(* IEC 61131-3 sources: RL_MAR/experiments/comparison/llm4plc/results/deepseek-ai-DeepSeek-V3.2_20260506_104945/20260506_120133, 4 files *)

(* ---- generated_code_iteration_0.st ---- *)
START_ST
FUNCTION_BLOCK CarParkingSystem
VAR_INPUT
    NewCarSlot : INT; (* Input for new car arrival slot number *)
END_VAR
VAR_OUTPUT
    Elevator1Busy : BOOL; (* Elevator 1 status - busy or idle *)
    Elevator2Busy : BOOL; (* Elevator 2 status - busy or idle *)
    Elevator1Position : INT; (* Elevator 1 current position *)
    Elevator2Position : INT; (* Elevator 2 current position *)
END_VAR
VAR
    Elevator1Target : INT; (* Elevator 1 target floor *)
    Elevator2Target : INT; (* Elevator 2 target floor *)
    CarSlots : ARRAY[1..100] OF BOOL; (* Array to represent parking slots - TRUE if occupied *)
    CurrentSlot : INT; (* Loop counter for scanning slots *)
    stateSys : INT; (* System state variable *)
    stateElev1 : INT; (* Elevator 1 state variable *)
    stateElev2 : INT; (* Elevator 2 state variable *)
    prevStateSys : INT; (* Previous system state for debugging or transitions *)
    prevStateElev1 : INT; (* Previous elevator 1 state *)
    prevStateElev2 : INT; (* Previous elevator 2 state *)
    tempSlot : INT; (* Temporary variable for processing new car slot *)
    movementStep : INT; (* Step size for elevator movement per cycle *)
    prevNewCarSlot : INT; (* Previous value of NewCarSlot for edge detection *)
    newArrivalDetected : BOOL; (* Flag to indicate a new arrival *)
    SYS_INIT : INT := 0; (* Constant for system initialization state *)
    SYS_SCAN : INT := 1; (* Constant for system scanning state *)
    ELEV_IDLE : INT := 0; (* Constant for elevator idle state *)
    ELEV_MOVING : INT := 1; (* Constant for elevator moving state *)
END_VAR

(* System state machine and elevator control logic *)
CASE stateSys OF
    SYS_INIT:
        (* Initialize all variables *)
        Elevator1Busy := FALSE;
        Elevator2Busy := FALSE;
        Elevator1Position := 0;
        Elevator2Position := 0;
        Elevator1Target := 0;
        Elevator2Target := 0;
        stateElev1 := ELEV_IDLE;
        stateElev2 := ELEV_IDLE;
        prevStateSys := SYS_INIT;
        prevStateElev1 := ELEV_IDLE;
        prevStateElev2 := ELEV_IDLE;
        tempSlot := 0;
        movementStep := 1;
        prevNewCarSlot := 0;
        newArrivalDetected := FALSE;
        FOR CurrentSlot := 1 TO 100 DO
            CarSlots[CurrentSlot] := FALSE;
        END_FOR;
        stateSys := SYS_SCAN; (* Transition to scanning state *)

    SYS_SCAN:
        (* Detect new car arrival by checking for change in NewCarSlot *)
        IF NewCarSlot <> prevNewCarSlot THEN
            newArrivalDetected := TRUE;
            prevNewCarSlot := NewCarSlot;
        ELSE
            newArrivalDetected := FALSE;
        END_IF;

        (* Process new arrival if detected and valid *)
        IF newArrivalDetected AND (NewCarSlot >= 1) AND (NewCarSlot <= 100) THEN
            IF NOT CarSlots[NewCarSlot] THEN
                CarSlots[NewCarSlot] := TRUE; (* Mark slot as occupied *)
                tempSlot := NewCarSlot;
                (* Assign target to appropriate elevator based on slot range *)
                IF (tempSlot >= 1) AND (tempSlot <= 50) THEN
                    (* Assign to Elevator 1 if idle *)
                    IF stateElev1 = ELEV_IDLE THEN
                        Elevator1Target := tempSlot;
                        stateElev1 := ELEV_MOVING;
                    END_IF;
                ELSIF (tempSlot >= 51) AND (tempSlot <= 100) THEN
                    (* Assign to Elevator 2 if idle *)
                    IF stateElev2 = ELEV_IDLE THEN
                        Elevator2Target := tempSlot;
                        stateElev2 := ELEV_MOVING;
                    END_IF;
                END_IF;
            END_IF;
        END_IF;

        (* Update Elevator 1 state and position *)
        CASE stateElev1 OF
            ELEV_IDLE:
                Elevator1Busy := FALSE;
                (* Position remains unchanged *)

            ELEV_MOVING:
                Elevator1Busy := TRUE;
                (* Move towards target by movementStep per cycle *)
                IF Elevator1Position < Elevator1Target THEN
                    Elevator1Position := Elevator1Position + movementStep;
                    IF Elevator1Position > Elevator1Target THEN
                        Elevator1Position := Elevator1Target;
                    END_IF;
                ELSIF Elevator1Position > Elevator1Target THEN
                    Elevator1Position := Elevator1Position - movementStep;
                    IF Elevator1Position < Elevator1Target THEN
                        Elevator1Position := Elevator1Target;
                    END_IF;
                END_IF;
                (* Check if target reached *)
                IF Elevator1Position = Elevator1Target THEN
                    stateElev1 := ELEV_IDLE;
                END_IF;
        END_CASE;

        (* Update Elevator 2 state and position *)
        CASE stateElev2 OF
            ELEV_IDLE:
                Elevator2Busy := FALSE;
                (* Position remains unchanged *)

            ELEV_MOVING:
                Elevator2Busy := TRUE;
                (* Move towards target by movementStep per cycle *)
                IF Elevator2Position < Elevator2Target THEN
                    Elevator2Position := Elevator2Position + movementStep;
                    IF Elevator2Position > Elevator2Target THEN
                        Elevator2Position := Elevator2Target;
                    END_IF;
                ELSIF Elevator2Position > Elevator2Target THEN
                    Elevator2Position := Elevator2Position - movementStep;
                    IF Elevator2Position < Elevator2Target THEN
                        Elevator2Position := Elevator2Target;
                    END_IF;
                END_IF;
                (* Check if target reached *)
                IF Elevator2Position = Elevator2Target THEN
                    stateElev2 := ELEV_IDLE;
                END_IF;
        END_CASE;

        (* Store previous states for potential debugging *)
        prevStateSys := stateSys;
        prevStateElev1 := stateElev1;
        prevStateElev2 := stateElev2;

        (* System remains in scanning state *)
        stateSys := SYS_SCAN;

END_CASE;

END_FUNCTION_BLOCK
END_ST

(* ---- generated_code_iteration_1.st ---- *)
START_REASON
The validation feedback indicates a CODESYS compiler error: "CASE标号要求文字或符号整型常量". This translates to "CASE label requires a literal or symbolic integer constant." This error occurs because in the provided ST code, the CASE statement for `stateSys` uses variables `SYS_INIT` and `SYS_SCAN` as case labels, but these are declared as variables within the VAR section with initial values (e.g., `SYS_INIT : INT := 0;`). In CODESYS, CASE labels must be constants (literals like 0, 1, or symbolic constants defined with `CONSTANT`), not variables. Variables cannot be used as case labels because their values can change at runtime, which is not allowed for case selection. To fix this, I need to declare `SYS_INIT`, `SYS_SCAN`, `ELEV_IDLE`, and `ELEV_MOVING` as constants using the `CONSTANT` keyword in a separate VAR_CONSTANT section, ensuring they are immutable and can be used as case labels. Additionally, I should ensure proper variable declarations and maintain the FUNCTION_BLOCK structure as required.
END_REASON

START_ST
FUNCTION_BLOCK CarParkingSystem
VAR_INPUT
    NewCarSlot : INT; (* Input for new car arrival slot number *)
END_VAR
VAR_OUTPUT
    Elevator1Busy : BOOL; (* Elevator 1 status - busy or idle *)
    Elevator2Busy : BOOL; (* Elevator 2 status - busy or idle *)
    Elevator1Position : INT; (* Elevator 1 current position *)
    Elevator2Position : INT; (* Elevator 2 current position *)
END_VAR
VAR
    Elevator1Target : INT; (* Elevator 1 target floor *)
    Elevator2Target : INT; (* Elevator 2 target floor *)
    CarSlots : ARRAY[1..100] OF BOOL; (* Array to represent parking slots - TRUE if occupied *)
    CurrentSlot : INT; (* Loop counter for scanning slots *)
    stateSys : INT; (* System state variable *)
    stateElev1 : INT; (* Elevator 1 state variable *)
    stateElev2 : INT; (* Elevator 2 state variable *)
    prevStateSys : INT; (* Previous system state for debugging or transitions *)
    prevStateElev1 : INT; (* Previous elevator 1 state *)
    prevStateElev2 : INT; (* Previous elevator 2 state *)
    tempSlot : INT; (* Temporary variable for processing new car slot *)
    movementStep : INT; (* Step size for elevator movement per cycle *)
    prevNewCarSlot : INT; (* Previous value of NewCarSlot for edge detection *)
    newArrivalDetected : BOOL; (* Flag to indicate a new arrival *)
END_VAR
VAR_CONSTANT
    SYS_INIT : INT := 0; (* Constant for system initialization state *)
    SYS_SCAN : INT := 1; (* Constant for system scanning state *)
    ELEV_IDLE : INT := 0; (* Constant for elevator idle state *)
    ELEV_MOVING : INT := 1; (* Constant for elevator moving state *)
END_VAR

(* System state machine and elevator control logic *)
CASE stateSys OF
    SYS_INIT:
        (* Initialize all variables *)
        Elevator1Busy := FALSE;
        Elevator2Busy := FALSE;
        Elevator1Position := 0;
        Elevator2Position := 0;
        Elevator1Target := 0;
        Elevator2Target := 0;
        stateElev1 := ELEV_IDLE;
        stateElev2 := ELEV_IDLE;
        prevStateSys := SYS_INIT;
        prevStateElev1 := ELEV_IDLE;
        prevStateElev2 := ELEV_IDLE;
        tempSlot := 0;
        movementStep := 1;
        prevNewCarSlot := 0;
        newArrivalDetected := FALSE;
        FOR CurrentSlot := 1 TO 100 DO
            CarSlots[CurrentSlot] := FALSE;
        END_FOR;
        stateSys := SYS_SCAN; (* Transition to scanning state *)

    SYS_SCAN:
        (* Detect new car arrival by checking for change in NewCarSlot *)
        IF NewCarSlot <> prevNewCarSlot THEN
            newArrivalDetected := TRUE;
            prevNewCarSlot := NewCarSlot;
        ELSE
            newArrivalDetected := FALSE;
        END_IF;

        (* Process new arrival if detected and valid *)
        IF newArrivalDetected AND (NewCarSlot >= 1) AND (NewCarSlot <= 100) THEN
            IF NOT CarSlots[NewCarSlot] THEN
                CarSlots[NewCarSlot] := TRUE; (* Mark slot as occupied *)
                tempSlot := NewCarSlot;
                (* Assign target to appropriate elevator based on slot range *)
                IF (tempSlot >= 1) AND (tempSlot <= 50) THEN
                    (* Assign to Elevator 1 if idle *)
                    IF stateElev1 = ELEV_IDLE THEN
                        Elevator1Target := tempSlot;
                        stateElev1 := ELEV_MOVING;
                    END_IF;
                ELSIF (tempSlot >= 51) AND (tempSlot <= 100) THEN
                    (* Assign to Elevator 2 if idle *)
                    IF stateElev2 = ELEV_IDLE THEN
                        Elevator2Target := tempSlot;
                        stateElev2 := ELEV_MOVING;
                    END_IF;
                END_IF;
            END_IF;
        END_IF;

        (* Update Elevator 1 state and position *)
        CASE stateElev1 OF
            ELEV_IDLE:
                Elevator1Busy := FALSE;
                (* Position remains unchanged *)

            ELEV_MOVING:
                Elevator1Busy := TRUE;
                (* Move towards target by movementStep per cycle *)
                IF Elevator1Position < Elevator1Target THEN
                    Elevator1Position := Elevator1Position + movementStep;
                    IF Elevator1Position > Elevator1Target THEN
                        Elevator1Position := Elevator1Target;
                    END_IF;
                ELSIF Elevator1Position > Elevator1Target THEN
                    Elevator1Position := Elevator1Position - movementStep;
                    IF Elevator1Position < Elevator1Target THEN
                        Elevator1Position := Elevator1Target;
                    END_IF;
                END_IF;
                (* Check if target reached *)
                IF Elevator1Position = Elevator1Target THEN
                    stateElev1 := ELEV_IDLE;
                END_IF;
        END_CASE;

        (* Update Elevator 2 state and position *)
        CASE stateElev2 OF
            ELEV_IDLE:
                Elevator2Busy := FALSE;
                (* Position remains unchanged *)

            ELEV_MOVING:
                Elevator2Busy := TRUE;
                (* Move towards target by movementStep per cycle *)
                IF Elevator2Position < Elevator2Target THEN
                    Elevator2Position := Elevator2Position + movementStep;
                    IF Elevator2Position > Elevator2Target THEN
                        Elevator2Position := Elevator2Target;
                    END_IF;
                ELSIF Elevator2Position > Elevator2Target THEN
                    Elevator2Position := Elevator2Position - movementStep;
                    IF Elevator2Position < Elevator2Target THEN
                        Elevator2Position := Elevator2Target;
                    END_IF;
                END_IF;
                (* Check if target reached *)
                IF Elevator2Position = Elevator2Target THEN
                    stateElev2 := ELEV_IDLE;
                END_IF;
        END_CASE;

        (* Store previous states for potential debugging *)
        prevStateSys := stateSys;
        prevStateElev1 := stateElev1;
        prevStateElev2 := stateElev2;

        (* System remains in scanning state *)
        stateSys := SYS_SCAN;

END_CASE;

END_FUNCTION_BLOCK
END_ST

(* ---- generated_code_iteration_2.st ---- *)
START_REASON
The validation feedback indicates an encoding issue: "gbk codec can't decode byte 0xac in position 101: illegal multibyte sequence." This suggests that the ST code contains a character that cannot be decoded with the GBK encoding, likely due to a special character like a non-breaking space, curly quotes, or an em dash that was inadvertently included. This could have been introduced in the previous response, possibly from copying or formatting. To fix this, I need to ensure the code uses only ASCII characters or properly encoded UTF-8 characters if supported, but for safety, I'll stick to basic ASCII characters (e.g., standard quotes, spaces, and alphanumeric symbols). I'll regenerate the code from scratch, ensuring no special or invisible characters are present, and maintain the FUNCTION_BLOCK structure with constants in VAR_CONSTANT as previously corrected. I'll also verify that all syntax is correct for CODESYS, including proper use of CASE statements with constants.
END_REASON

START_ST
FUNCTION_BLOCK CarParkingSystem
VAR_INPUT
    NewCarSlot : INT; (* Input for new car arrival slot number *)
END_VAR
VAR_OUTPUT
    Elevator1Busy : BOOL; (* Elevator 1 status - busy or idle *)
    Elevator2Busy : BOOL; (* Elevator 2 status - busy or idle *)
    Elevator1Position : INT; (* Elevator 1 current position *)
    Elevator2Position : INT; (* Elevator 2 current position *)
END_VAR
VAR
    Elevator1Target : INT; (* Elevator 1 target floor *)
    Elevator2Target : INT; (* Elevator 2 target floor *)
    CarSlots : ARRAY[1..100] OF BOOL; (* Array to represent parking slots - TRUE if occupied *)
    CurrentSlot : INT; (* Loop counter for scanning slots *)
    stateSys : INT; (* System state variable *)
    stateElev1 : INT; (* Elevator 1 state variable *)
    stateElev2 : INT; (* Elevator 2 state variable *)
    prevStateSys : INT; (* Previous system state for debugging or transitions *)
    prevStateElev1 : INT; (* Previous elevator 1 state *)
    prevStateElev2 : INT; (* Previous elevator 2 state *)
    tempSlot : INT; (* Temporary variable for processing new car slot *)
    movementStep : INT; (* Step size for elevator movement per cycle *)
    prevNewCarSlot : INT; (* Previous value of NewCarSlot for edge detection *)
    newArrivalDetected : BOOL; (* Flag to indicate a new arrival *)
END_VAR
VAR_CONSTANT
    SYS_INIT : INT := 0; (* Constant for system initialization state *)
    SYS_SCAN : INT := 1; (* Constant for system scanning state *)
    ELEV_IDLE : INT := 0; (* Constant for elevator idle state *)
    ELEV_MOVING : INT := 1; (* Constant for elevator moving state *)
END_VAR

(* System state machine and elevator control logic *)
CASE stateSys OF
    SYS_INIT:
        (* Initialize all variables *)
        Elevator1Busy := FALSE;
        Elevator2Busy := FALSE;
        Elevator1Position := 0;
        Elevator2Position := 0;
        Elevator1Target := 0;
        Elevator2Target := 0;
        stateElev1 := ELEV_IDLE;
        stateElev2 := ELEV_IDLE;
        prevStateSys := SYS_INIT;
        prevStateElev1 := ELEV_IDLE;
        prevStateElev2 := ELEV_IDLE;
        tempSlot := 0;
        movementStep := 1;
        prevNewCarSlot := 0;
        newArrivalDetected := FALSE;
        FOR CurrentSlot := 1 TO 100 DO
            CarSlots[CurrentSlot] := FALSE;
        END_FOR;
        stateSys := SYS_SCAN; (* Transition to scanning state *)

    SYS_SCAN:
        (* Detect new car arrival by checking for change in NewCarSlot *)
        IF NewCarSlot <> prevNewCarSlot THEN
            newArrivalDetected := TRUE;
            prevNewCarSlot := NewCarSlot;
        ELSE
            newArrivalDetected := FALSE;
        END_IF;

        (* Process new arrival if detected and valid *)
        IF newArrivalDetected AND (NewCarSlot >= 1) AND (NewCarSlot <= 100) THEN
            IF NOT CarSlots[NewCarSlot] THEN
                CarSlots[NewCarSlot] := TRUE; (* Mark slot as occupied *)
                tempSlot := NewCarSlot;
                (* Assign target to appropriate elevator based on slot range *)
                IF (tempSlot >= 1) AND (tempSlot <= 50) THEN
                    (* Assign to Elevator 1 if idle *)
                    IF stateElev1 = ELEV_IDLE THEN
                        Elevator1Target := tempSlot;
                        stateElev1 := ELEV_MOVING;
                    END_IF;
                ELSIF (tempSlot >= 51) AND (tempSlot <= 100) THEN
                    (* Assign to Elevator 2 if idle *)
                    IF stateElev2 = ELEV_IDLE THEN
                        Elevator2Target := tempSlot;
                        stateElev2 := ELEV_MOVING;
                    END_IF;
                END_IF;
            END_IF;
        END_IF;

        (* Update Elevator 1 state and position *)
        CASE stateElev1 OF
            ELEV_IDLE:
                Elevator1Busy := FALSE;
                (* Position remains unchanged *)

            ELEV_MOVING:
                Elevator1Busy := TRUE;
                (* Move towards target by movementStep per cycle *)
                IF Elevator1Position < Elevator1Target THEN
                    Elevator1Position := Elevator1Position + movementStep;
                    IF Elevator1Position > Elevator1Target THEN
                        Elevator1Position := Elevator1Target;
                    END_IF;
                ELSIF Elevator1Position > Elevator1Target THEN
                    Elevator1Position := Elevator1Position - movementStep;
                    IF Elevator1Position < Elevator1Target THEN
                        Elevator1Position := Elevator1Target;
                    END_IF;
                END_IF;
                (* Check if target reached *)
                IF Elevator1Position = Elevator1Target THEN
                    stateElev1 := ELEV_IDLE;
                END_IF;
        END_CASE;

        (* Update Elevator 2 state and position *)
        CASE stateElev2 OF
            ELEV_IDLE:
                Elevator2Busy := FALSE;
                (* Position remains unchanged *)

            ELEV_MOVING:
                Elevator2Busy := TRUE;
                (* Move towards target by movementStep per cycle *)
                IF Elevator2Position < Elevator2Target THEN
                    Elevator2Position := Elevator2Position + movementStep;
                    IF Elevator2Position > Elevator2Target THEN
                        Elevator2Position := Elevator2Target;
                    END_IF;
                ELSIF Elevator2Position > Elevator2Target THEN
                    Elevator2Position := Elevator2Position - movementStep;
                    IF Elevator2Position < Elevator2Target THEN
                        Elevator2Position := Elevator2Target;
                    END_IF;
                END_IF;
                (* Check if target reached *)
                IF Elevator2Position = Elevator2Target THEN
                    stateElev2 := ELEV_IDLE;
                END_IF;
        END_CASE;

        (* Store previous states for potential debugging *)
        prevStateSys := stateSys;
        prevStateElev1 := stateElev1;
        prevStateElev2 := stateElev2;

        (* System remains in scanning state *)
        stateSys := SYS_SCAN;

END_CASE;

END_FUNCTION_BLOCK
END_ST

(* ---- generated_code_iteration_3.st ---- *)
START_REASON
The validation feedback indicates a CODESYS compiler error: "应该采用VAR, VAR_INPUT, VAR_OUTPUT 或 VAR_IN_OUT 取代VAR_CONSTANT:;" which translates to "Should use VAR, VAR_INPUT, VAR_OUTPUT or VAR_IN_OUT instead of VAR_CONSTANT:;". This suggests that in the CODESYS environment, the VAR_CONSTANT section is not recognized or is syntactically incorrect. In CODESYS Structured Text, constants should be declared within the VAR section using the CONSTANT keyword, not in a separate VAR_CONSTANT block. I need to replace VAR_CONSTANT with VAR CONSTANT to make it compliant with CODESYS syntax. Additionally, I'll ensure all other syntax elements are correct, such as proper variable declarations and CASE statements. I'll regenerate the code with this correction, maintaining the FUNCTION_BLOCK structure and all required logic.
END_REASON

START_ST
FUNCTION_BLOCK CarParkingSystem
VAR_INPUT
    NewCarSlot : INT; (* Input for new car arrival slot number *)
END_VAR
VAR_OUTPUT
    Elevator1Busy : BOOL; (* Elevator 1 status - busy or idle *)
    Elevator2Busy : BOOL; (* Elevator 2 status - busy or idle *)
    Elevator1Position : INT; (* Elevator 1 current position *)
    Elevator2Position : INT; (* Elevator 2 current position *)
END_VAR
VAR
    Elevator1Target : INT; (* Elevator 1 target floor *)
    Elevator2Target : INT; (* Elevator 2 target floor *)
    CarSlots : ARRAY[1..100] OF BOOL; (* Array to represent parking slots - TRUE if occupied *)
    CurrentSlot : INT; (* Loop counter for scanning slots *)
    stateSys : INT; (* System state variable *)
    stateElev1 : INT; (* Elevator 1 state variable *)
    stateElev2 : INT; (* Elevator 2 state variable *)
    prevStateSys : INT; (* Previous system state for debugging or transitions *)
    prevStateElev1 : INT; (* Previous elevator 1 state *)
    prevStateElev2 : INT; (* Previous elevator 2 state *)
    tempSlot : INT; (* Temporary variable for processing new car slot *)
    movementStep : INT; (* Step size for elevator movement per cycle *)
    prevNewCarSlot : INT; (* Previous value of NewCarSlot for edge detection *)
    newArrivalDetected : BOOL; (* Flag to indicate a new arrival *)
END_VAR
VAR CONSTANT
    SYS_INIT : INT := 0; (* Constant for system initialization state *)
    SYS_SCAN : INT := 1; (* Constant for system scanning state *)
    ELEV_IDLE : INT := 0; (* Constant for elevator idle state *)
    ELEV_MOVING : INT := 1; (* Constant for elevator moving state *)
END_VAR

(* System state machine and elevator control logic *)
CASE stateSys OF
    SYS_INIT:
        (* Initialize all variables *)
        Elevator1Busy := FALSE;
        Elevator2Busy := FALSE;
        Elevator1Position := 0;
        Elevator2Position := 0;
        Elevator1Target := 0;
        Elevator2Target := 0;
        stateElev1 := ELEV_IDLE;
        stateElev2 := ELEV_IDLE;
        prevStateSys := SYS_INIT;
        prevStateElev1 := ELEV_IDLE;
        prevStateElev2 := ELEV_IDLE;
        tempSlot := 0;
        movementStep := 1;
        prevNewCarSlot := 0;
        newArrivalDetected := FALSE;
        FOR CurrentSlot := 1 TO 100 DO
            CarSlots[CurrentSlot] := FALSE;
        END_FOR;
        stateSys := SYS_SCAN; (* Transition to scanning state *)

    SYS_SCAN:
        (* Detect new car arrival by checking for change in NewCarSlot *)
        IF NewCarSlot <> prevNewCarSlot THEN
            newArrivalDetected := TRUE;
            prevNewCarSlot := NewCarSlot;
        ELSE
            newArrivalDetected := FALSE;
        END_IF;

        (* Process new arrival if detected and valid *)
        IF newArrivalDetected AND (NewCarSlot >= 1) AND (NewCarSlot <= 100) THEN
            IF NOT CarSlots[NewCarSlot] THEN
                CarSlots[NewCarSlot] := TRUE; (* Mark slot as occupied *)
                tempSlot := NewCarSlot;
                (* Assign target to appropriate elevator based on slot range *)
                IF (tempSlot >= 1) AND (tempSlot <= 50) THEN
                    (* Assign to Elevator 1 if idle *)
                    IF stateElev1 = ELEV_IDLE THEN
                        Elevator1Target := tempSlot;
                        stateElev1 := ELEV_MOVING;
                    END_IF;
                ELSIF (tempSlot >= 51) AND (tempSlot <= 100) THEN
                    (* Assign to Elevator 2 if idle *)
                    IF stateElev2 = ELEV_IDLE THEN
                        Elevator2Target := tempSlot;
                        stateElev2 := ELEV_MOVING;
                    END_IF;
                END_IF;
            END_IF;
        END_IF;

        (* Update Elevator 1 state and position *)
        CASE stateElev1 OF
            ELEV_IDLE:
                Elevator1Busy := FALSE;
                (* Position remains unchanged *)

            ELEV_MOVING:
                Elevator1Busy := TRUE;
                (* Move towards target by movementStep per cycle *)
                IF Elevator1Position < Elevator1Target THEN
                    Elevator1Position := Elevator1Position + movementStep;
                    IF Elevator1Position > Elevator1Target THEN
                        Elevator1Position := Elevator1Target;
                    END_IF;
                ELSIF Elevator1Position > Elevator1Target THEN
                    Elevator1Position := Elevator1Position - movementStep;
                    IF Elevator1Position < Elevator1Target THEN
                        Elevator1Position := Elevator1Target;
                    END_IF;
                END_IF;
                (* Check if target reached *)
                IF Elevator1Position = Elevator1Target THEN
                    stateElev1 := ELEV_IDLE;
                END_IF;
        END_CASE;

        (* Update Elevator 2 state and position *)
        CASE stateElev2 OF
            ELEV_IDLE:
                Elevator2Busy := FALSE;
                (* Position remains unchanged *)

            ELEV_MOVING:
                Elevator2Busy := TRUE;
                (* Move towards target by movementStep per cycle *)
                IF Elevator2Position < Elevator2Target THEN
                    Elevator2Position := Elevator2Position + movementStep;
                    IF Elevator2Position > Elevator2Target THEN
                        Elevator2Position := Elevator2Target;
                    END_IF;
                ELSIF Elevator2Position > Elevator2Target THEN
                    Elevator2Position := Elevator2Position - movementStep;
                    IF Elevator2Position < Elevator2Target THEN
                        Elevator2Position := Elevator2Target;
                    END_IF;
                END_IF;
                (* Check if target reached *)
                IF Elevator2Position = Elevator2Target THEN
                    stateElev2 := ELEV_IDLE;
                END_IF;
        END_CASE;

        (* Store previous states for potential debugging *)
        prevStateSys := stateSys;
        prevStateElev1 := stateElev1;
        prevStateElev2 := stateElev2;

        (* System remains in scanning state *)
        stateSys := SYS_SCAN;

END_CASE;

END_FUNCTION_BLOCK
END_ST
